// TIA Portal V16 export
// export: Created 2023-03-29T11:04:47.4490964Z, ExportSetting WithDefaults, DisplayName Totally Integrated Automation Portal, DisplayVersion V16 Update 6, DisplayName TIA Portal Version Control Interface, DisplayVersion V16 Update 2, DisplayName TIA Portal Openness, DisplayVersion V16 Update 6, DisplayName STEP 7 Professional, DisplayVersion V16 Update 6, DisplayName STEP 7 Safety, DisplayVersion V16, DisplayName WinCC Advanced, DisplayVersion V16 Update 6
FUNCTION "Wybór_pompy_najmniej godzin" : Void   // FC17, LAD
TITLE = Selektor godzin pracy / Compressor selection from hours
{ S7_Optimized_Access := 'TRUE' }
AUTHOR : rtecmer
VERSION : 0.1
// Ustawienie kolejności wyboru pomp z wyrównaniem czasu pracy. Podstawa najmniejsza ilość godzin pracy / Ustawienie kolejności wyboru kompresorów z wyrównaniem czasu pracy. Podstawa najmniejsza ilość godzin pracy
// stored: AutoNumber true, IsIECCheckEnabled false, SetENOAutomatically false, UDAEnableTagReadback false
   VAR_IN_OUT
      Reset : Bool;   // Reset po błędzie
   END_VAR
   VAR_TEMP
      tmp_Sum_sek_P1 : Int;   // tymczasowy licznik sumy sekund
      tmp_Sum_sek_P2 : Int;   // tymczasowy licznik sumy sekund
      tmp_Sum_sek_P3 : Int;   // tymczasowy licznik sumy sekund
      tmp_Sum_sek_P4 : Int;   // tymczasowy licznik sumy sekund
   END_VAR
BEGIN

REGION Network 1: Reakcja na równe liczniki
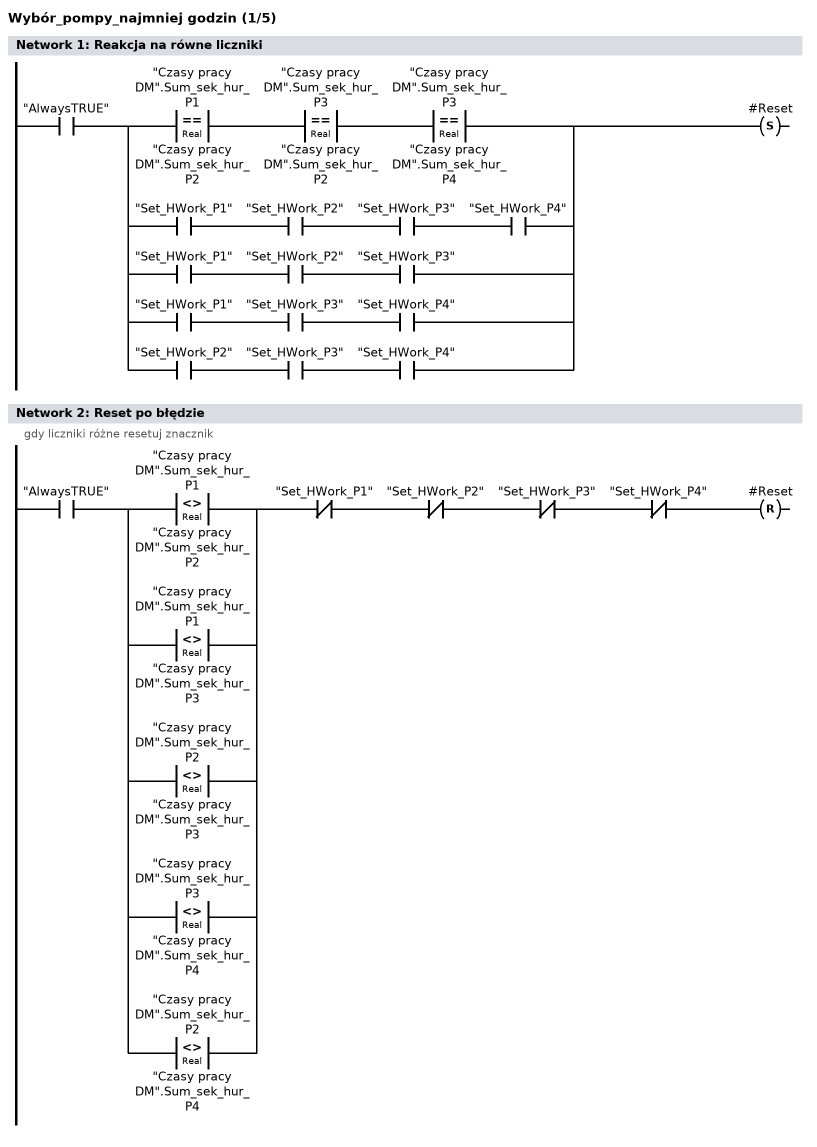
   RUNG wire#powerrail
      Contact( "AlwaysTRUE" )
      wire#w1
      { S7_Templates := "SrcType := Real" } EQ_Contact(in1 := "Czasy pracy DM".Sum_sek_hur_P1, in2 := "Czasy pracy DM".Sum_sek_hur_P2)
      { S7_Templates := "SrcType := Real" } EQ_Contact(in1 := "Czasy pracy DM".Sum_sek_hur_P3, in2 := "Czasy pracy DM".Sum_sek_hur_P2)
      { S7_Templates := "SrcType := Real" } EQ_Contact(in1 := "Czasy pracy DM".Sum_sek_hur_P3, in2 := "Czasy pracy DM".Sum_sek_hur_P4)
      wire#w2
      S_Coil( #Reset )
   END_RUNG
   RUNG wire#w1
      Contact( "Set_HWork_P1" )
      Contact( "Set_HWork_P2" )
      Contact( "Set_HWork_P3" )
      Contact( "Set_HWork_P4" )
   END_RUNG wire#w2
   RUNG wire#w1
      Contact( "Set_HWork_P1" )
      Contact( "Set_HWork_P2" )
      Contact( "Set_HWork_P3" )
   END_RUNG wire#w2
   RUNG wire#w1
      Contact( "Set_HWork_P1" )
      Contact( "Set_HWork_P3" )
      Contact( "Set_HWork_P4" )
   END_RUNG wire#w2
   RUNG wire#w1
      Contact( "Set_HWork_P2" )
      Contact( "Set_HWork_P3" )
      Contact( "Set_HWork_P4" )
   END_RUNG wire#w2
   // the same network as SCL:
   IF "AlwaysTRUE" AND ((("Czasy pracy DM".Sum_sek_hur_P1 = "Czasy pracy DM".Sum_sek_hur_P2) AND ("Czasy pracy DM".Sum_sek_hur_P3 = "Czasy pracy DM".Sum_sek_hur_P2) AND ("Czasy pracy DM".Sum_sek_hur_P3 = "Czasy pracy DM".Sum_sek_hur_P4)) OR ("Set_HWork_P1" AND "Set_HWork_P2" AND "Set_HWork_P3" AND "Set_HWork_P4") OR ("Set_HWork_P1" AND "Set_HWork_P2" AND "Set_HWork_P3") OR ("Set_HWork_P1" AND "Set_HWork_P3" AND "Set_HWork_P4") OR ("Set_HWork_P2" AND "Set_HWork_P3" AND "Set_HWork_P4")) THEN
       #Reset := TRUE;
   END_IF;
END_REGION

REGION Network 2: Reset po błędzie
   // gdy liczniki różne resetuj znacznik
   RUNG wire#powerrail
      Contact( "AlwaysTRUE" )
      wire#w1
      { S7_Templates := "SrcType := Real" } NE_Contact(in1 := "Czasy pracy DM".Sum_sek_hur_P1, in2 := "Czasy pracy DM".Sum_sek_hur_P2)
      wire#w2
      I_Contact( "Set_HWork_P1" )
      I_Contact( "Set_HWork_P2" )
      I_Contact( "Set_HWork_P3" )
      I_Contact( "Set_HWork_P4" )
      R_Coil( #Reset )
   END_RUNG
   RUNG wire#w1
      { S7_Templates := "SrcType := Real" } NE_Contact(in1 := "Czasy pracy DM".Sum_sek_hur_P1, in2 := "Czasy pracy DM".Sum_sek_hur_P3)
   END_RUNG wire#w2
   RUNG wire#w1
      { S7_Templates := "SrcType := Real" } NE_Contact(in1 := "Czasy pracy DM".Sum_sek_hur_P2, in2 := "Czasy pracy DM".Sum_sek_hur_P3)
   END_RUNG wire#w2
   RUNG wire#w1
      { S7_Templates := "SrcType := Real" } NE_Contact(in1 := "Czasy pracy DM".Sum_sek_hur_P3, in2 := "Czasy pracy DM".Sum_sek_hur_P4)
   END_RUNG wire#w2
   RUNG wire#w1
      { S7_Templates := "SrcType := Real" } NE_Contact(in1 := "Czasy pracy DM".Sum_sek_hur_P2, in2 := "Czasy pracy DM".Sum_sek_hur_P4)
   END_RUNG wire#w2
   // the same network as SCL:
   IF "AlwaysTRUE" AND (("Czasy pracy DM".Sum_sek_hur_P1 <> "Czasy pracy DM".Sum_sek_hur_P2) OR ("Czasy pracy DM".Sum_sek_hur_P1 <> "Czasy pracy DM".Sum_sek_hur_P3) OR ("Czasy pracy DM".Sum_sek_hur_P2 <> "Czasy pracy DM".Sum_sek_hur_P3) OR ("Czasy pracy DM".Sum_sek_hur_P3 <> "Czasy pracy DM".Sum_sek_hur_P4) OR ("Czasy pracy DM".Sum_sek_hur_P2 <> "Czasy pracy DM".Sum_sek_hur_P4)) AND NOT "Set_HWork_P1" AND NOT "Set_HWork_P2" AND NOT "Set_HWork_P3" AND NOT "Set_HWork_P4" THEN
       #Reset := FALSE;
   END_IF;
END_REGION

REGION Network 3: Reset znaczników aktywacji napędu od czasu pracy / Wyłączenie napedów od równych liczników
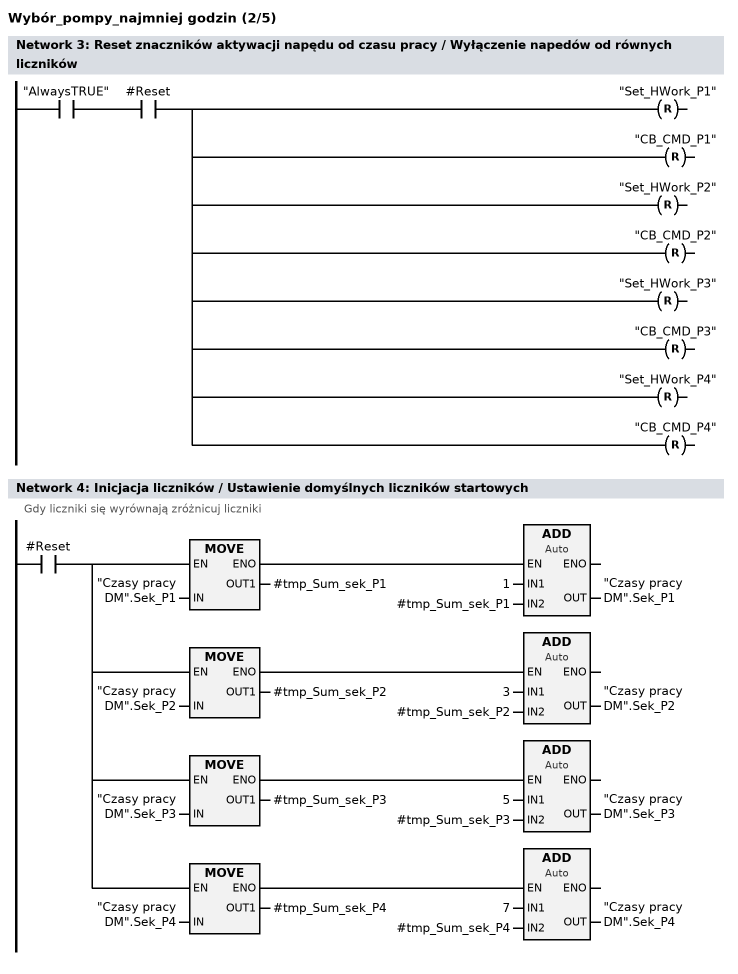
   RUNG wire#powerrail
      Contact( "AlwaysTRUE" )
      Contact( #Reset )
      wire#w1
      R_Coil( "Set_HWork_P1" )
   END_RUNG
   RUNG wire#w1
      R_Coil( "CB_CMD_P1" )
   END_RUNG
   RUNG wire#w1
      R_Coil( "Set_HWork_P2" )
   END_RUNG
   RUNG wire#w1
      R_Coil( "CB_CMD_P2" )
   END_RUNG
   RUNG wire#w1
      R_Coil( "Set_HWork_P3" )
   END_RUNG
   RUNG wire#w1
      R_Coil( "CB_CMD_P3" )
   END_RUNG
   RUNG wire#w1
      R_Coil( "Set_HWork_P4" )
   END_RUNG
   RUNG wire#w1
      R_Coil( "CB_CMD_P4" )
   END_RUNG
   // the same network as SCL:
   IF "AlwaysTRUE" AND #Reset THEN
       "Set_HWork_P1" := FALSE;
       "CB_CMD_P1" := FALSE;
       "Set_HWork_P2" := FALSE;
       "CB_CMD_P2" := FALSE;
       "Set_HWork_P3" := FALSE;
       "CB_CMD_P3" := FALSE;
       "Set_HWork_P4" := FALSE;
       "CB_CMD_P4" := FALSE;
   END_IF;
END_REGION

REGION Network 4: Inicjacja liczników / Ustawienie domyślnych liczników startowych
   // Gdy liczniki się wyrównają zróżnicuj liczniki
   RUNG wire#powerrail
      Contact( #Reset )
      wire#w1
      Move(in := "Czasy pracy DM".Sek_P1, out1 => #tmp_Sum_sek_P1)
      Add(in1 := 1, in2 := #tmp_Sum_sek_P1, out => "Czasy pracy DM".Sek_P1)
   END_RUNG
   RUNG wire#w1
      Move(in := "Czasy pracy DM".Sek_P2, out1 => #tmp_Sum_sek_P2)
      Add(in1 := 3, in2 := #tmp_Sum_sek_P2, out => "Czasy pracy DM".Sek_P2)
   END_RUNG
   RUNG wire#w1
      Move(in := "Czasy pracy DM".Sek_P3, out1 => #tmp_Sum_sek_P3)
      Add(in1 := 5, in2 := #tmp_Sum_sek_P3, out => "Czasy pracy DM".Sek_P3)
   END_RUNG
   RUNG wire#w1
      Move(in := "Czasy pracy DM".Sek_P4, out1 => #tmp_Sum_sek_P4)
      Add(in1 := 7, in2 := #tmp_Sum_sek_P4, out => "Czasy pracy DM".Sek_P4)
   END_RUNG
   // the same network as SCL:
   IF #Reset THEN
       #tmp_Sum_sek_P1 := "Czasy pracy DM".Sek_P1;
       "Czasy pracy DM".Sek_P1 := 1 + #tmp_Sum_sek_P1;
       #tmp_Sum_sek_P2 := "Czasy pracy DM".Sek_P2;
       "Czasy pracy DM".Sek_P2 := 3 + #tmp_Sum_sek_P2;
       #tmp_Sum_sek_P3 := "Czasy pracy DM".Sek_P3;
       "Czasy pracy DM".Sek_P3 := 5 + #tmp_Sum_sek_P3;
       #tmp_Sum_sek_P4 := "Czasy pracy DM".Sek_P4;
       "Czasy pracy DM".Sek_P4 := 7 + #tmp_Sum_sek_P4;
   END_IF;
END_REGION

REGION Network 5: Znacznik wyrównywania czasu pracy z falownika P1 / Znacznik wyrównywania czasu pracy z falownika dla P1
   // %DB10.DBX7.7 - bit tryb automat M7
   // Jesli najmniej godzin pracy to usta znacznik.
   // Ale bierz pod uwagę czy kompresor P2 , P3 już nie pracuje lub nie jest w trybie automat.
   // bit tryb automat P1
   // Jesli najmniej godzin pracy to usta znacznik.
   // Ale bierz po uwagę czy kompresor P1 , P4 już nie pracuje lub nie jest w trybie automat.
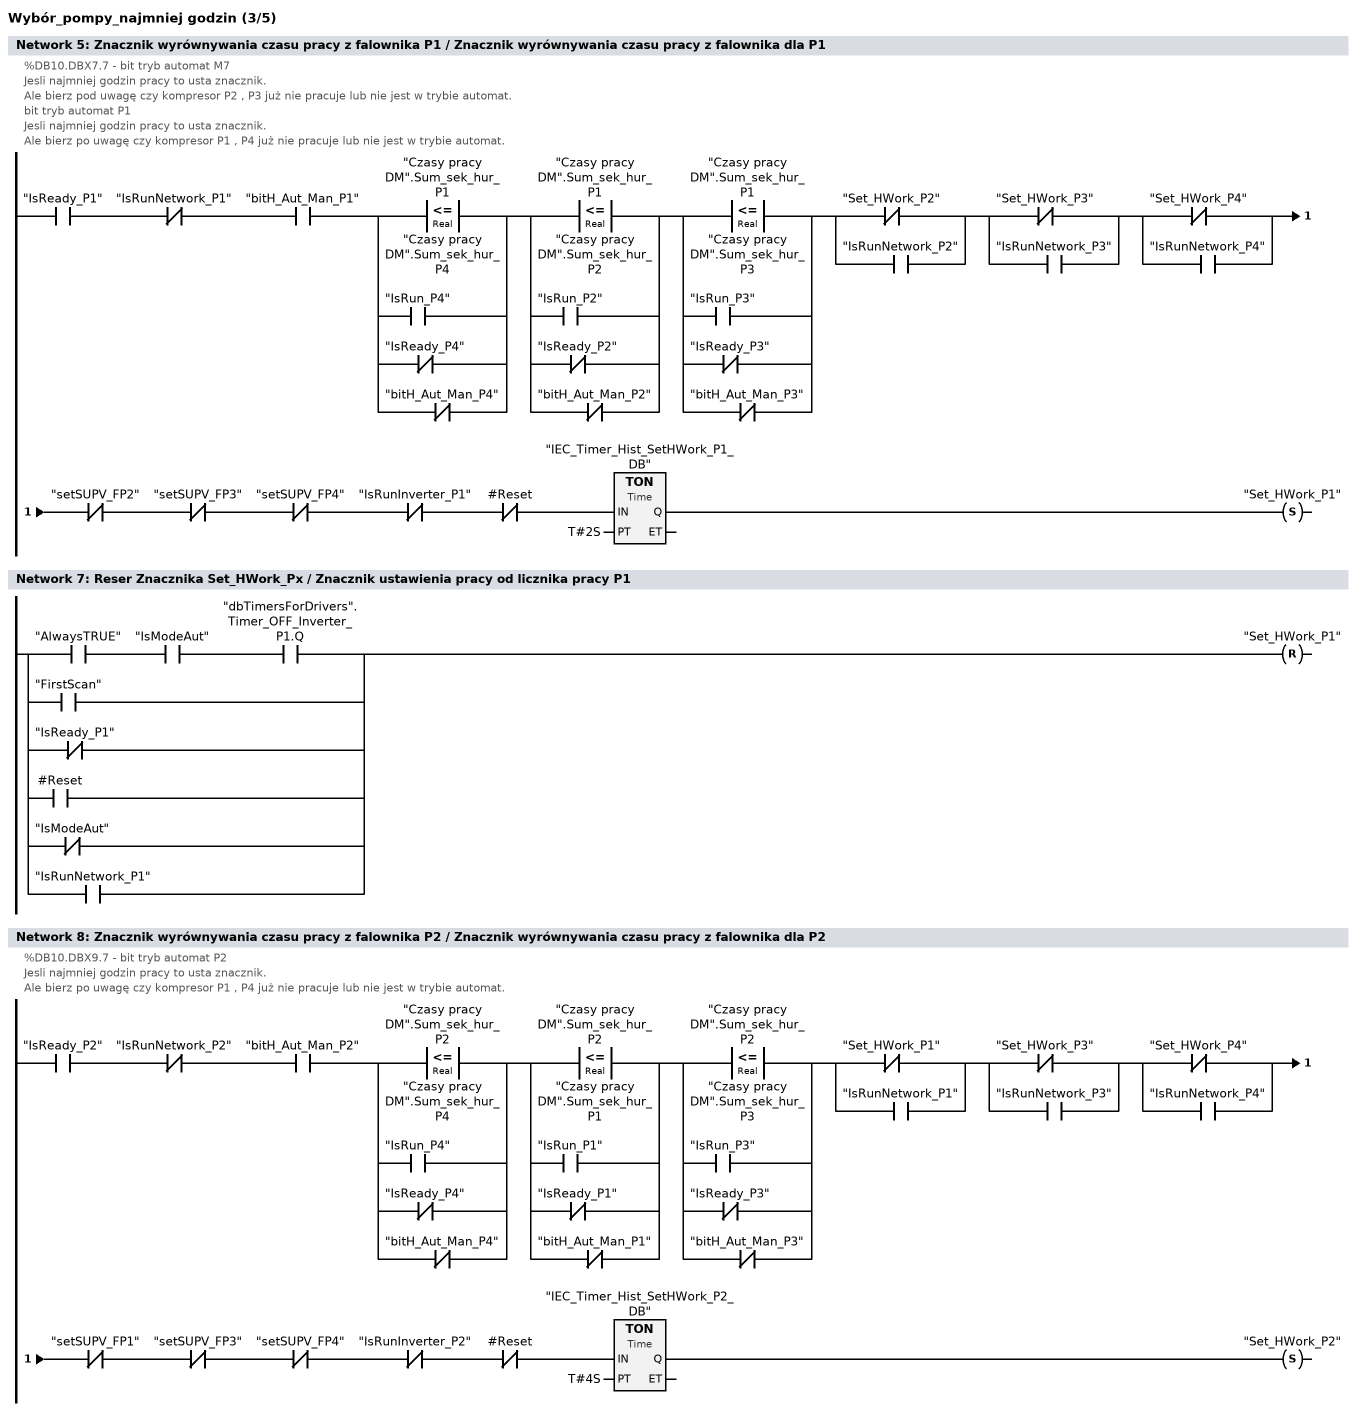
   RUNG wire#powerrail
      Contact( "IsReady_P1" )
      I_Contact( "IsRunNetwork_P1" )
      Contact( "bitH_Aut_Man_P1" )
      wire#w1
      { S7_Templates := "SrcType := Real" } LE_Contact(in1 := "Czasy pracy DM".Sum_sek_hur_P1, in2 := "Czasy pracy DM".Sum_sek_hur_P4)
      wire#w2
      { S7_Templates := "SrcType := Real" } LE_Contact(in1 := "Czasy pracy DM".Sum_sek_hur_P1, in2 := "Czasy pracy DM".Sum_sek_hur_P2)
      wire#w3
      { S7_Templates := "SrcType := Real" } LE_Contact(in1 := "Czasy pracy DM".Sum_sek_hur_P1, in2 := "Czasy pracy DM".Sum_sek_hur_P3)
      wire#w4
      I_Contact( "Set_HWork_P2" )
      wire#w5
      I_Contact( "Set_HWork_P3" )
      wire#w6
      I_Contact( "Set_HWork_P4" )
      wire#w7
      I_Contact( "setSUPV_FP2" )
      I_Contact( "setSUPV_FP3" )
      I_Contact( "setSUPV_FP4" )
      I_Contact( "IsRunInverter_P1" )
      I_Contact( #Reset )
      { S7_Templates := "time_type := Time" } "IEC_Timer_Hist_SetHWork_P1_DB".TON(pt := T#2S, et =>)
      S_Coil( "Set_HWork_P1" )
   END_RUNG
   RUNG wire#w1
      Contact( "IsRun_P4" )
   END_RUNG wire#w2
   RUNG wire#w1
      I_Contact( "IsReady_P4" )
   END_RUNG wire#w2
   RUNG wire#w1
      I_Contact( "bitH_Aut_Man_P4" )
   END_RUNG wire#w2
   RUNG wire#w2
      Contact( "IsRun_P2" )
   END_RUNG wire#w3
   RUNG wire#w2
      I_Contact( "IsReady_P2" )
   END_RUNG wire#w3
   RUNG wire#w2
      I_Contact( "bitH_Aut_Man_P2" )
   END_RUNG wire#w3
   RUNG wire#w3
      Contact( "IsRun_P3" )
   END_RUNG wire#w4
   RUNG wire#w3
      I_Contact( "IsReady_P3" )
   END_RUNG wire#w4
   RUNG wire#w3
      I_Contact( "bitH_Aut_Man_P3" )
   END_RUNG wire#w4
   RUNG wire#w4
      Contact( "IsRunNetwork_P2" )
   END_RUNG wire#w5
   RUNG wire#w5
      Contact( "IsRunNetwork_P3" )
   END_RUNG wire#w6
   RUNG wire#w6
      Contact( "IsRunNetwork_P4" )
   END_RUNG wire#w7
   // the same network as SCL:
   "IEC_Timer_Hist_SetHWork_P1_DB".TON(IN := "IsReady_P1" AND NOT "IsRunNetwork_P1" AND "bitH_Aut_Man_P1" AND (("Czasy pracy DM".Sum_sek_hur_P1 <= "Czasy pracy DM".Sum_sek_hur_P4) OR "IsRun_P4" OR NOT "IsReady_P4" OR NOT "bitH_Aut_Man_P4") AND (("Czasy pracy DM".Sum_sek_hur_P1 <= "Czasy pracy DM".Sum_sek_hur_P2) OR "IsRun_P2" OR NOT "IsReady_P2" OR NOT "bitH_Aut_Man_P2") AND (("Czasy pracy DM".Sum_sek_hur_P1 <= "Czasy pracy DM".Sum_sek_hur_P3) OR "IsRun_P3" OR NOT "IsReady_P3" OR NOT "bitH_Aut_Man_P3") AND (NOT "Set_HWork_P2" OR "IsRunNetwork_P2") AND (NOT "Set_HWork_P3" OR "IsRunNetwork_P3") AND (NOT "Set_HWork_P4" OR "IsRunNetwork_P4") AND NOT "setSUPV_FP2" AND NOT "setSUPV_FP3" AND NOT "setSUPV_FP4" AND NOT "IsRunInverter_P1" AND NOT #Reset,
                           PT := T#2S);
   IF "IEC_Timer_Hist_SetHWork_P1_DB".Q THEN "Set_HWork_P1" := TRUE; END_IF;
END_REGION

REGION Network 6 (SCL): Sprawdzanie czy aktywna w trybie AUT
   IF "Set_HWork_P1" = TRUE AND "bitH_Aut_Man_P1" = FALSE THEN
     // Statement section IF
     "Set_HWork_P1" := FALSE;
     ;
   END_IF;
END_REGION

REGION Network 7: Reser Znacznika Set_HWork_Px / Znacznik ustawienia pracy od licznika pracy P1
   RUNG wire#powerrail
      Contact( "AlwaysTRUE" )
      Contact( "IsModeAut" )
      Contact( "dbTimersForDrivers".Timer_OFF_Inverter_P1.Q )
      wire#w1
      R_Coil( "Set_HWork_P1" )
   END_RUNG
   RUNG wire#powerrail
      Contact( "FirstScan" )
   END_RUNG wire#w1
   RUNG wire#powerrail
      I_Contact( "IsReady_P1" )
   END_RUNG wire#w1
   RUNG wire#powerrail
      Contact( #Reset )
   END_RUNG wire#w1
   RUNG wire#powerrail
      I_Contact( "IsModeAut" )
   END_RUNG wire#w1
   RUNG wire#powerrail
      Contact( "IsRunNetwork_P1" )
   END_RUNG wire#w1
   // the same network as SCL:
   IF ("AlwaysTRUE" AND "IsModeAut" AND "dbTimersForDrivers".Timer_OFF_Inverter_P1.Q) OR "FirstScan" OR NOT "IsReady_P1" OR #Reset OR NOT "IsModeAut" OR "IsRunNetwork_P1" THEN
       "Set_HWork_P1" := FALSE;
   END_IF;
END_REGION

REGION Network 8: Znacznik wyrównywania czasu pracy z falownika P2 / Znacznik wyrównywania czasu pracy z falownika dla P2
   // %DB10.DBX9.7 - bit tryb automat P2
   // Jesli najmniej godzin pracy to usta znacznik.
   // Ale bierz po uwagę czy kompresor P1 , P4 już nie pracuje lub nie jest w trybie automat.
   RUNG wire#powerrail
      Contact( "IsReady_P2" )
      I_Contact( "IsRunNetwork_P2" )
      Contact( "bitH_Aut_Man_P2" )
      wire#w1
      { S7_Templates := "SrcType := Real" } LE_Contact(in1 := "Czasy pracy DM".Sum_sek_hur_P2, in2 := "Czasy pracy DM".Sum_sek_hur_P4)
      wire#w2
      { S7_Templates := "SrcType := Real" } LE_Contact(in1 := "Czasy pracy DM".Sum_sek_hur_P2, in2 := "Czasy pracy DM".Sum_sek_hur_P1)
      wire#w3
      { S7_Templates := "SrcType := Real" } LE_Contact(in1 := "Czasy pracy DM".Sum_sek_hur_P2, in2 := "Czasy pracy DM".Sum_sek_hur_P3)
      wire#w4
      I_Contact( "Set_HWork_P1" )
      wire#w5
      I_Contact( "Set_HWork_P3" )
      wire#w6
      I_Contact( "Set_HWork_P4" )
      wire#w7
      I_Contact( "setSUPV_FP1" )
      I_Contact( "setSUPV_FP3" )
      I_Contact( "setSUPV_FP4" )
      I_Contact( "IsRunInverter_P2" )
      I_Contact( #Reset )
      { S7_Templates := "time_type := Time" } "IEC_Timer_Hist_SetHWork_P2_DB".TON(pt := T#4S, et =>)
      S_Coil( "Set_HWork_P2" )
   END_RUNG
   RUNG wire#w1
      Contact( "IsRun_P4" )
   END_RUNG wire#w2
   RUNG wire#w1
      I_Contact( "IsReady_P4" )
   END_RUNG wire#w2
   RUNG wire#w1
      I_Contact( "bitH_Aut_Man_P4" )
   END_RUNG wire#w2
   RUNG wire#w2
      Contact( "IsRun_P1" )
   END_RUNG wire#w3
   RUNG wire#w2
      I_Contact( "IsReady_P1" )
   END_RUNG wire#w3
   RUNG wire#w2
      I_Contact( "bitH_Aut_Man_P1" )
   END_RUNG wire#w3
   RUNG wire#w3
      Contact( "IsRun_P3" )
   END_RUNG wire#w4
   RUNG wire#w3
      I_Contact( "IsReady_P3" )
   END_RUNG wire#w4
   RUNG wire#w3
      I_Contact( "bitH_Aut_Man_P3" )
   END_RUNG wire#w4
   RUNG wire#w4
      Contact( "IsRunNetwork_P1" )
   END_RUNG wire#w5
   RUNG wire#w5
      Contact( "IsRunNetwork_P3" )
   END_RUNG wire#w6
   RUNG wire#w6
      Contact( "IsRunNetwork_P4" )
   END_RUNG wire#w7
   // the same network as SCL:
   "IEC_Timer_Hist_SetHWork_P2_DB".TON(IN := "IsReady_P2" AND NOT "IsRunNetwork_P2" AND "bitH_Aut_Man_P2" AND (("Czasy pracy DM".Sum_sek_hur_P2 <= "Czasy pracy DM".Sum_sek_hur_P4) OR "IsRun_P4" OR NOT "IsReady_P4" OR NOT "bitH_Aut_Man_P4") AND (("Czasy pracy DM".Sum_sek_hur_P2 <= "Czasy pracy DM".Sum_sek_hur_P1) OR "IsRun_P1" OR NOT "IsReady_P1" OR NOT "bitH_Aut_Man_P1") AND (("Czasy pracy DM".Sum_sek_hur_P2 <= "Czasy pracy DM".Sum_sek_hur_P3) OR "IsRun_P3" OR NOT "IsReady_P3" OR NOT "bitH_Aut_Man_P3") AND (NOT "Set_HWork_P1" OR "IsRunNetwork_P1") AND (NOT "Set_HWork_P3" OR "IsRunNetwork_P3") AND (NOT "Set_HWork_P4" OR "IsRunNetwork_P4") AND NOT "setSUPV_FP1" AND NOT "setSUPV_FP3" AND NOT "setSUPV_FP4" AND NOT "IsRunInverter_P2" AND NOT #Reset,
                           PT := T#4S);
   IF "IEC_Timer_Hist_SetHWork_P2_DB".Q THEN "Set_HWork_P2" := TRUE; END_IF;
END_REGION

REGION Network 9 (SCL): Sprawdzanie czy aktywna w trybie AUT
   IF "Set_HWork_P2" = TRUE AND "bitH_Aut_Man_P2" = FALSE THEN
     // Statement section IF
     "Set_HWork_P2" := FALSE;
     ;
   END_IF;
END_REGION

REGION Network 10: Reser Znacznika Set_HWork_Px / Znacznik ustawienia pracy od licznika pracy P2
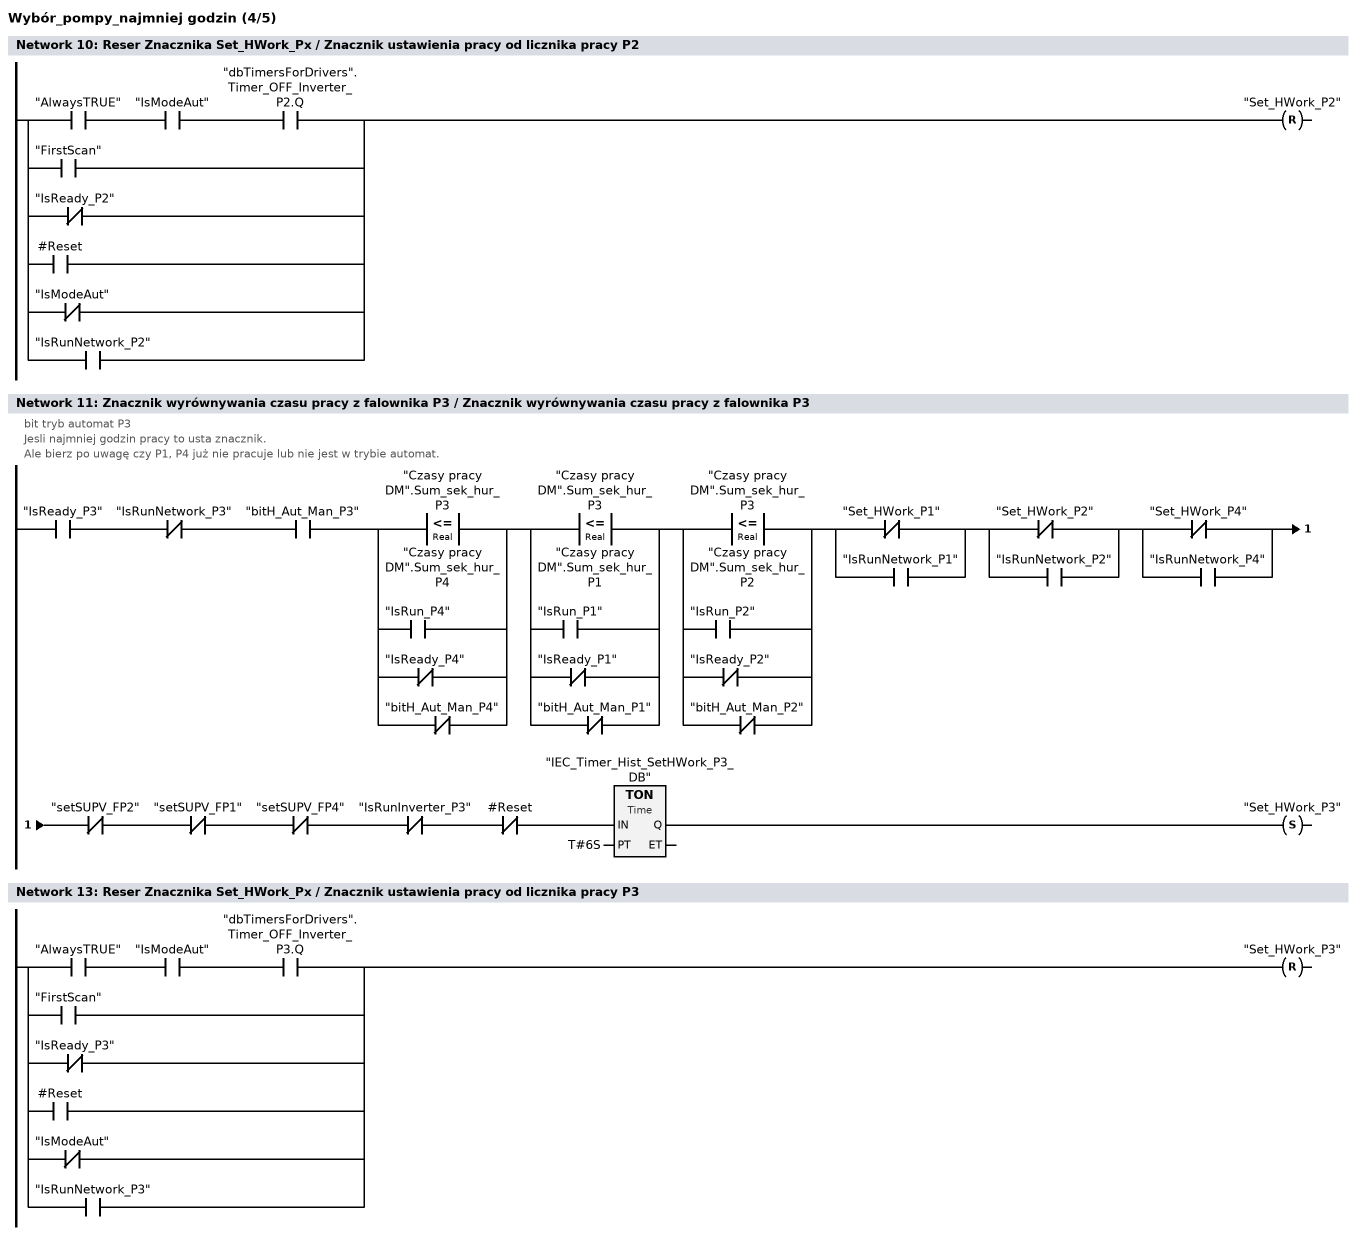
   RUNG wire#powerrail
      Contact( "AlwaysTRUE" )
      Contact( "IsModeAut" )
      Contact( "dbTimersForDrivers".Timer_OFF_Inverter_P2.Q )
      wire#w1
      R_Coil( "Set_HWork_P2" )
   END_RUNG
   RUNG wire#powerrail
      Contact( "FirstScan" )
   END_RUNG wire#w1
   RUNG wire#powerrail
      I_Contact( "IsReady_P2" )
   END_RUNG wire#w1
   RUNG wire#powerrail
      Contact( #Reset )
   END_RUNG wire#w1
   RUNG wire#powerrail
      I_Contact( "IsModeAut" )
   END_RUNG wire#w1
   RUNG wire#powerrail
      Contact( "IsRunNetwork_P2" )
   END_RUNG wire#w1
   // the same network as SCL:
   IF ("AlwaysTRUE" AND "IsModeAut" AND "dbTimersForDrivers".Timer_OFF_Inverter_P2.Q) OR "FirstScan" OR NOT "IsReady_P2" OR #Reset OR NOT "IsModeAut" OR "IsRunNetwork_P2" THEN
       "Set_HWork_P2" := FALSE;
   END_IF;
END_REGION

REGION Network 11: Znacznik wyrównywania czasu pracy z falownika P3 / Znacznik wyrównywania czasu pracy z falownika P3
   // bit tryb automat P3
   // Jesli najmniej godzin pracy to usta znacznik.
   // Ale bierz po uwagę czy P1, P4 już nie pracuje lub nie jest w trybie automat.
   RUNG wire#powerrail
      Contact( "IsReady_P3" )
      I_Contact( "IsRunNetwork_P3" )
      Contact( "bitH_Aut_Man_P3" )
      wire#w1
      { S7_Templates := "SrcType := Real" } LE_Contact(in1 := "Czasy pracy DM".Sum_sek_hur_P3, in2 := "Czasy pracy DM".Sum_sek_hur_P4)
      wire#w2
      { S7_Templates := "SrcType := Real" } LE_Contact(in1 := "Czasy pracy DM".Sum_sek_hur_P3, in2 := "Czasy pracy DM".Sum_sek_hur_P1)
      wire#w3
      { S7_Templates := "SrcType := Real" } LE_Contact(in1 := "Czasy pracy DM".Sum_sek_hur_P3, in2 := "Czasy pracy DM".Sum_sek_hur_P2)
      wire#w4
      I_Contact( "Set_HWork_P1" )
      wire#w5
      I_Contact( "Set_HWork_P2" )
      wire#w6
      I_Contact( "Set_HWork_P4" )
      wire#w7
      I_Contact( "setSUPV_FP2" )
      I_Contact( "setSUPV_FP1" )
      I_Contact( "setSUPV_FP4" )
      I_Contact( "IsRunInverter_P3" )
      I_Contact( #Reset )
      { S7_Templates := "time_type := Time" } "IEC_Timer_Hist_SetHWork_P3_DB".TON(pt := T#6S, et =>)
      S_Coil( "Set_HWork_P3" )
   END_RUNG
   RUNG wire#w1
      Contact( "IsRun_P4" )
   END_RUNG wire#w2
   RUNG wire#w1
      I_Contact( "IsReady_P4" )
   END_RUNG wire#w2
   RUNG wire#w1
      I_Contact( "bitH_Aut_Man_P4" )
   END_RUNG wire#w2
   RUNG wire#w2
      Contact( "IsRun_P1" )
   END_RUNG wire#w3
   RUNG wire#w2
      I_Contact( "IsReady_P1" )
   END_RUNG wire#w3
   RUNG wire#w2
      I_Contact( "bitH_Aut_Man_P1" )
   END_RUNG wire#w3
   RUNG wire#w3
      Contact( "IsRun_P2" )
   END_RUNG wire#w4
   RUNG wire#w3
      I_Contact( "IsReady_P2" )
   END_RUNG wire#w4
   RUNG wire#w3
      I_Contact( "bitH_Aut_Man_P2" )
   END_RUNG wire#w4
   RUNG wire#w4
      Contact( "IsRunNetwork_P1" )
   END_RUNG wire#w5
   RUNG wire#w5
      Contact( "IsRunNetwork_P2" )
   END_RUNG wire#w6
   RUNG wire#w6
      Contact( "IsRunNetwork_P4" )
   END_RUNG wire#w7
   // the same network as SCL:
   "IEC_Timer_Hist_SetHWork_P3_DB".TON(IN := "IsReady_P3" AND NOT "IsRunNetwork_P3" AND "bitH_Aut_Man_P3" AND (("Czasy pracy DM".Sum_sek_hur_P3 <= "Czasy pracy DM".Sum_sek_hur_P4) OR "IsRun_P4" OR NOT "IsReady_P4" OR NOT "bitH_Aut_Man_P4") AND (("Czasy pracy DM".Sum_sek_hur_P3 <= "Czasy pracy DM".Sum_sek_hur_P1) OR "IsRun_P1" OR NOT "IsReady_P1" OR NOT "bitH_Aut_Man_P1") AND (("Czasy pracy DM".Sum_sek_hur_P3 <= "Czasy pracy DM".Sum_sek_hur_P2) OR "IsRun_P2" OR NOT "IsReady_P2" OR NOT "bitH_Aut_Man_P2") AND (NOT "Set_HWork_P1" OR "IsRunNetwork_P1") AND (NOT "Set_HWork_P2" OR "IsRunNetwork_P2") AND (NOT "Set_HWork_P4" OR "IsRunNetwork_P4") AND NOT "setSUPV_FP2" AND NOT "setSUPV_FP1" AND NOT "setSUPV_FP4" AND NOT "IsRunInverter_P3" AND NOT #Reset,
                           PT := T#6S);
   IF "IEC_Timer_Hist_SetHWork_P3_DB".Q THEN "Set_HWork_P3" := TRUE; END_IF;
END_REGION

REGION Network 12 (SCL): Sprawdzanie czy aktywna w trybie AUT
   IF "Set_HWork_P3" = TRUE AND "bitH_Aut_Man_P3" = FALSE THEN
     // Statement section IF
     "Set_HWork_P3" := FALSE;
     ;
   END_IF;
END_REGION

REGION Network 13: Reser Znacznika Set_HWork_Px / Znacznik ustawienia pracy od licznika pracy P3
   RUNG wire#powerrail
      Contact( "AlwaysTRUE" )
      Contact( "IsModeAut" )
      Contact( "dbTimersForDrivers".Timer_OFF_Inverter_P3.Q )
      wire#w1
      R_Coil( "Set_HWork_P3" )
   END_RUNG
   RUNG wire#powerrail
      Contact( "FirstScan" )
   END_RUNG wire#w1
   RUNG wire#powerrail
      I_Contact( "IsReady_P3" )
   END_RUNG wire#w1
   RUNG wire#powerrail
      Contact( #Reset )
   END_RUNG wire#w1
   RUNG wire#powerrail
      I_Contact( "IsModeAut" )
   END_RUNG wire#w1
   RUNG wire#powerrail
      Contact( "IsRunNetwork_P3" )
   END_RUNG wire#w1
   // the same network as SCL:
   IF ("AlwaysTRUE" AND "IsModeAut" AND "dbTimersForDrivers".Timer_OFF_Inverter_P3.Q) OR "FirstScan" OR NOT "IsReady_P3" OR #Reset OR NOT "IsModeAut" OR "IsRunNetwork_P3" THEN
       "Set_HWork_P3" := FALSE;
   END_IF;
END_REGION

REGION Network 14: Znacznik wyrównywania czasu pracy z falownika P4 / Znacznik wyrównywania czasu pracy z falownika P4
   // bit tryb automat P4
   // Jesli najmniej godzin pracy to usta znacznik.
   // Ale bierz po uwagę czy P1, P4 już nie pracuje lub nie jest w trybie automat.
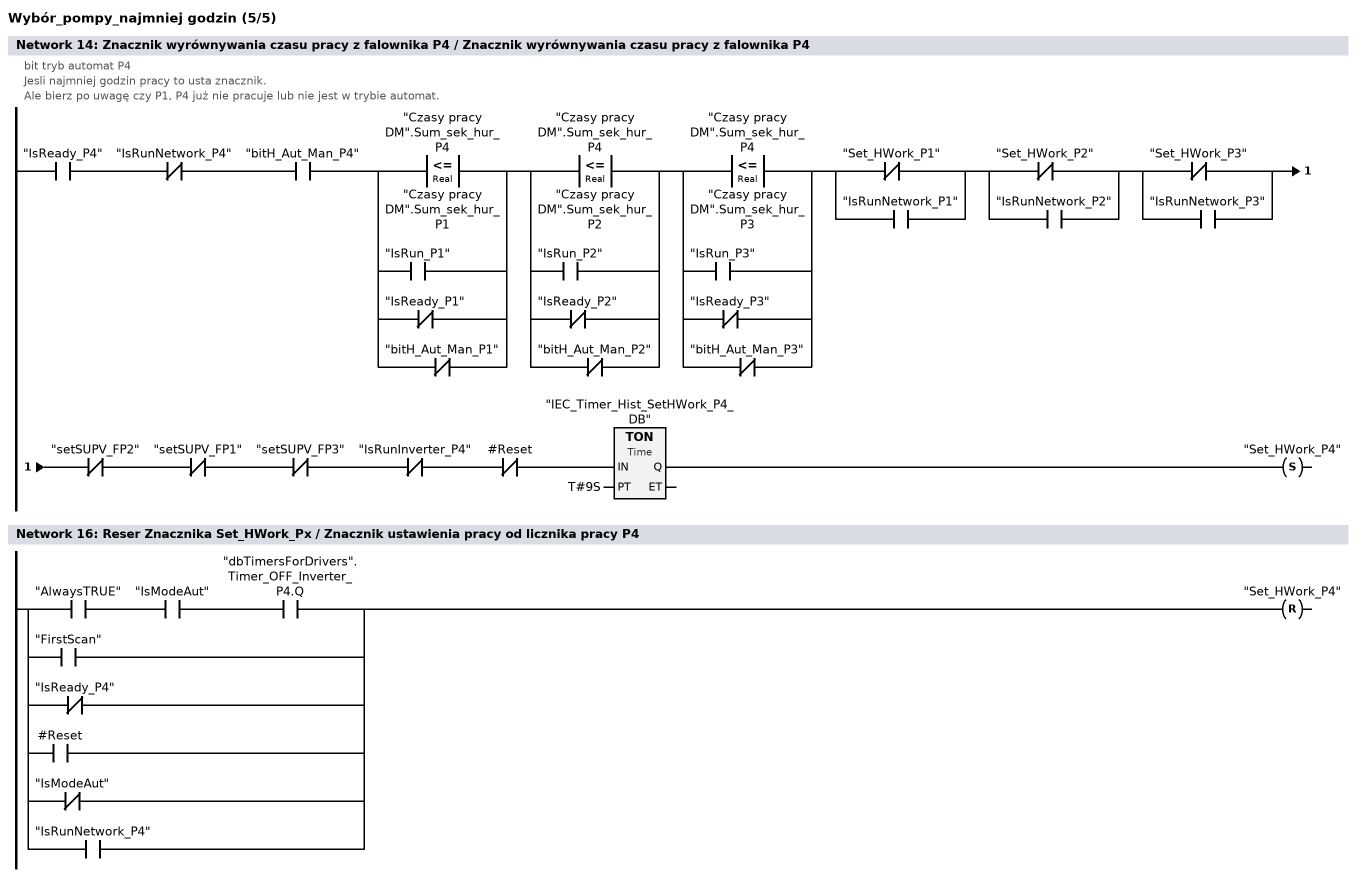
   RUNG wire#powerrail
      Contact( "IsReady_P4" )
      I_Contact( "IsRunNetwork_P4" )
      Contact( "bitH_Aut_Man_P4" )
      wire#w1
      { S7_Templates := "SrcType := Real" } LE_Contact(in1 := "Czasy pracy DM".Sum_sek_hur_P4, in2 := "Czasy pracy DM".Sum_sek_hur_P1)
      wire#w2
      { S7_Templates := "SrcType := Real" } LE_Contact(in1 := "Czasy pracy DM".Sum_sek_hur_P4, in2 := "Czasy pracy DM".Sum_sek_hur_P2)
      wire#w3
      { S7_Templates := "SrcType := Real" } LE_Contact(in1 := "Czasy pracy DM".Sum_sek_hur_P4, in2 := "Czasy pracy DM".Sum_sek_hur_P3)
      wire#w4
      I_Contact( "Set_HWork_P1" )
      wire#w5
      I_Contact( "Set_HWork_P2" )
      wire#w6
      I_Contact( "Set_HWork_P3" )
      wire#w7
      I_Contact( "setSUPV_FP2" )
      I_Contact( "setSUPV_FP1" )
      I_Contact( "setSUPV_FP3" )
      I_Contact( "IsRunInverter_P4" )
      I_Contact( #Reset )
      { S7_Templates := "time_type := Time" } "IEC_Timer_Hist_SetHWork_P4_DB".TON(pt := T#9S, et =>)
      S_Coil( "Set_HWork_P4" )
   END_RUNG
   RUNG wire#w1
      Contact( "IsRun_P1" )
   END_RUNG wire#w2
   RUNG wire#w1
      I_Contact( "IsReady_P1" )
   END_RUNG wire#w2
   RUNG wire#w1
      I_Contact( "bitH_Aut_Man_P1" )
   END_RUNG wire#w2
   RUNG wire#w2
      Contact( "IsRun_P2" )
   END_RUNG wire#w3
   RUNG wire#w2
      I_Contact( "IsReady_P2" )
   END_RUNG wire#w3
   RUNG wire#w2
      I_Contact( "bitH_Aut_Man_P2" )
   END_RUNG wire#w3
   RUNG wire#w3
      Contact( "IsRun_P3" )
   END_RUNG wire#w4
   RUNG wire#w3
      I_Contact( "IsReady_P3" )
   END_RUNG wire#w4
   RUNG wire#w3
      I_Contact( "bitH_Aut_Man_P3" )
   END_RUNG wire#w4
   RUNG wire#w4
      Contact( "IsRunNetwork_P1" )
   END_RUNG wire#w5
   RUNG wire#w5
      Contact( "IsRunNetwork_P2" )
   END_RUNG wire#w6
   RUNG wire#w6
      Contact( "IsRunNetwork_P3" )
   END_RUNG wire#w7
   // the same network as SCL:
   "IEC_Timer_Hist_SetHWork_P4_DB".TON(IN := "IsReady_P4" AND NOT "IsRunNetwork_P4" AND "bitH_Aut_Man_P4" AND (("Czasy pracy DM".Sum_sek_hur_P4 <= "Czasy pracy DM".Sum_sek_hur_P1) OR "IsRun_P1" OR NOT "IsReady_P1" OR NOT "bitH_Aut_Man_P1") AND (("Czasy pracy DM".Sum_sek_hur_P4 <= "Czasy pracy DM".Sum_sek_hur_P2) OR "IsRun_P2" OR NOT "IsReady_P2" OR NOT "bitH_Aut_Man_P2") AND (("Czasy pracy DM".Sum_sek_hur_P4 <= "Czasy pracy DM".Sum_sek_hur_P3) OR "IsRun_P3" OR NOT "IsReady_P3" OR NOT "bitH_Aut_Man_P3") AND (NOT "Set_HWork_P1" OR "IsRunNetwork_P1") AND (NOT "Set_HWork_P2" OR "IsRunNetwork_P2") AND (NOT "Set_HWork_P3" OR "IsRunNetwork_P3") AND NOT "setSUPV_FP2" AND NOT "setSUPV_FP1" AND NOT "setSUPV_FP3" AND NOT "IsRunInverter_P4" AND NOT #Reset,
                           PT := T#9S);
   IF "IEC_Timer_Hist_SetHWork_P4_DB".Q THEN "Set_HWork_P4" := TRUE; END_IF;
END_REGION

REGION Network 15 (SCL): Sprawdzanie czy aktywna w trybie AUT
   IF "Set_HWork_P4" = TRUE AND "bitH_Aut_Man_P4" = FALSE THEN
     // Statement section IF
     "Set_HWork_P4" := FALSE;
     ;
   END_IF;
END_REGION

REGION Network 16: Reser Znacznika Set_HWork_Px / Znacznik ustawienia pracy od licznika pracy P4
   RUNG wire#powerrail
      Contact( "AlwaysTRUE" )
      Contact( "IsModeAut" )
      Contact( "dbTimersForDrivers".Timer_OFF_Inverter_P4.Q )
      wire#w1
      R_Coil( "Set_HWork_P4" )
   END_RUNG
   RUNG wire#powerrail
      Contact( "FirstScan" )
   END_RUNG wire#w1
   RUNG wire#powerrail
      I_Contact( "IsReady_P4" )
   END_RUNG wire#w1
   RUNG wire#powerrail
      Contact( #Reset )
   END_RUNG wire#w1
   RUNG wire#powerrail
      I_Contact( "IsModeAut" )
   END_RUNG wire#w1
   RUNG wire#powerrail
      Contact( "IsRunNetwork_P4" )
   END_RUNG wire#w1
   // the same network as SCL:
   IF ("AlwaysTRUE" AND "IsModeAut" AND "dbTimersForDrivers".Timer_OFF_Inverter_P4.Q) OR "FirstScan" OR NOT "IsReady_P4" OR #Reset OR NOT "IsModeAut" OR "IsRunNetwork_P4" THEN
       "Set_HWork_P4" := FALSE;
   END_IF;
END_REGION
END_FUNCTION
